{attribute addProperty BoxType "EK1122-0000-0018"}
{attribute addProperty Id "Beckhoff_EL31xxsub_EK1100EK1100_179A0949162"}
{attribute addProperty CRC "4082504356"}
{attribute addProperty SizeInBites "16"}
{attribute addProperty SizeInBytes "2"}
TYPE Beckhoff_EL31xxEK1122_F35612A4 EXTENDS EK1122_179A0949 :
STRUCT
	{attribute addProperty Name "Beckhoff_EL31xxsub_EK1100"}
	Beckhoff_EL31xxsub_EK1100 : EK1100_179A0949;
END_STRUCT
END_TYPE

(* stored: Version 1.2.0.0, ProductVersion 3.1.4024.9
   DUT Beckhoff_EL31xxEK1122_F35612A4: Id {d0b3329b-a58c-4396-852c-0f2bafd895e2} *)
